PROGRAM MAIN
VAR
	step : INT := 0;
	
	Count : int := 0;
END_VAR

CASE step OF
	0:
		IF Data_In.AxisPosUse[Count] THEN
			SendDataFrame.Send(Data_In.AxisPos[Count], Count);
			step := step + 1;
		END_IF
		
		Count := Count + 1;
		IF Count > 15 THEN
			Count := 0;
		END_IF
		
	1:
		IF NOT SendDataFrame.bDone THEN
			step := step + 1;
		END_IF
		
	2:
		IF SendDataFrame.bDone THEN
			step := 0;
		END_IF
END_CASE

SendDataFrame();

END_PROGRAM

(* stored: Version 1.1.0.1, ProductVersion 3.1.4024.15
   POU MAIN: Id {c78d8a4c-bb7a-42a5-be73-6c75da82ad3b}, SpecialFunc None *)
